# EPICS autosave request: iocBoot/ioc13Keithley1/auto_settings.req
file "Keithley2kDMM_mf22_settings.req", P=13Keithley1:, Dmm=DMM1
file "scan_settings.req",               P=13Keithley1:, S=scan1
file "scan_settings.req",               P=13Keithley1:, S=scan2
file "scan_settings.req",               P=13Keithley1:, S=scan3
file "scan_settings.req",               P=13Keithley1:, S=scan4
